// TIA Portal V17 export
VAR_GLOBAL   // PLC tag table "HMI"
   StartCmd AT %I0.0 : Bool;   // HMI start pushbutton
   StopCmd AT %I0.1 : Bool;   // HMI stop pushbutton (NC)
END_VAR
